PROGRAM MAIN
VAR
END_VAR

END_PROGRAM

(* stored: Version 1.1.0.1
   POU MAIN: Id {452f7adb-2ae3-42f1-8cb2-ca6582b1099e} *)
